Fanuc KAREL source: NC0088.KL

PROGRAM NC0088
%NOLOCKGROUP
ROUTINE R
VAR
S1:INTEGER;S2:INTEGER;S3:INTEGER;S4:INTEGER
BEGIN
--
--
--
S1=1
IF (S1=1) THEN
SELECT S1 OF
CASE(1):
FOR S2=1 TO 2 DO
WHILE (S1<2) DO
IF (S1=1) THEN
SELECT S1 OF
CASE(1):
FOR S3=1 TO 2 DO
WHILE (S1<2) DO
IF (S1=1) THEN
SELECT S1 OF
CASE(1):
FOR S4=1 TO 2 DO
WHILE (S1<2) DO
S1=(S1+1)
ENDWHILE
ENDFOR
CASE(2):
S1=(S1+2)
ELSE:
S1=(S1+3)
ENDSELECT
ELSE
S1=(S1+2)
ENDIF
ENDWHILE
ENDFOR
CASE(2):
S1=(S1+2)
ELSE:
S1=(S1+3)
ENDSELECT
ELSE
S1=(S1+2)
ENDIF
ENDWHILE
ENDFOR
CASE(2):
S1=(S1+2)
ELSE:
S1=(S1+3)
ENDSELECT
ELSE
S1=(S1+2)
ENDIF
END R
BEGIN
R
END NC0088
